// TIA Portal V18 export
// export: Created 2025-12-01T12:39:35.9184725Z, ExportSetting None, DisplayName Totally Integrated Automation Portal, DisplayVersion V18 Update 5, DisplayName TIA Portal Openness, DisplayVersion V18 Update 5, DisplayName TIA Portal Teamcenter Gateway, DisplayVersion V18, DisplayName TIA Portal Version Control Interface, DisplayVersion V18, DisplayName STEP 7 Professional, DisplayVersion V18 Update 5, DisplayName STEP 7 Safety, DisplayVersion V18, DisplayName WinCC Professional, DisplayVersion V18 Update 5
VAR_GLOBAL   // PLC tag table "PartType"
END_VAR
VAR_GLOBAL CONSTANT   // user constants
   PartTypeFor_11KW : USInt := 1;
   PartTypeFor_22KW : USInt := 2;
   Cy10GoHome : UInt := 0;
   Cy10GoWork : UInt := 1;
END_VAR
